// TwinCAT 3 PLC project Tc_Math
// Title: Tc_Math
// Company: NewEngineer
// Author: https://github.com/phucpha
// ProjectVersion: 0.0.0.1
// Description: this is library expand the Tc2_math
// ProgramVersion: 3.1.4024.0
// libraries:
//   Tc2_Standard, * (Beckhoff Automation GmbH)
//   Tc2_System, * (Beckhoff Automation GmbH)
//   Tc2_Utilities, * (Beckhoff Automation GmbH)
//   Tc3_Module, * (Beckhoff Automation GmbH)
// project tree:
//   DUTs/ E_CompareTime.TcDUT (not stored)
//   FCs/ F_CompareTime.TcPOU (not stored), FUN_Ceil.TcPOU (not stored), F_CheckInRange.TcPOU (not stored), F_CubicFit.TcPOU (not stored), F_CubitCalculate.TcPOU (not stored), F_InRange.TcPOU, F_QuanDraticCalculate.TcPOU (not stored), F_QuandraticFomularMaxValue.TcPOU (not stored), F_RoundLrealEx.TcPOU (not stored), F_ScaleValue.TcPOU (not stored)
//   / PlcTask.TcTTO (not stored)
//   POUs/ FB_CalCulateAccumulation.TcPOU (not stored), FB_Derivative.TcPOU

// ---- FCs/F_InRange.TcPOU
FUNCTION F_InRange : BOOL // return true if value in [bound1, bound2] or in [bound2, bound1] else return false
VAR_INPUT
	bound1 : LREAL;
	bound2 : LREAL;
	value	: LREAL;
END_VAR
VAR
END_VAR

F_InRange := (MIN(bound1, bound2) <= value)
				AND (value <= MAX(bound1, bound2));

END_FUNCTION

// ---- POUs/FB_Derivative.TcPOU
(*algorithm: Backward differentiation formula
the higher other the less stable , but more accuracy*)
FUNCTION_BLOCK FB_Derivative// unit : dentalvalue/seconde
VAR_INPUT
	bReset : BOOL	:= FALSE; //BOOL //reset
	lrInputValue : LREAL;// actual function value
	tDerivative	: TIME	:= T#1S; //length of time interval [tn−1,tn]  (equals time passed since last call to function)
	nOrder		: UINT := 3;// The s-step or order in algorithm // recommend
END_VAR
VAR_OUTPUT
	lrDerivative : LREAL;
	xValid : BOOL;//Validity OF result FALSE: If the number of calls neccessary for approximating has not been executed yet.
END_VAR
VAR
	ftn :LREAL;
	ftn_1 : LREAL;
	ftn_2 : LREAL;
	ftn_3 : LREAL;
	ftn_4 : LREAL;
	ftn_5	: LREAL;
	ftn_6	: LREAL;
	tonUpdate : TON;
	nTimeUpdate : LREAL;
END_VAR

IF bReset THEN
	tonUpdate.IN := FALSE;
	ftn := 0 ;
	ftn_1 := 0;
	ftn_2 := 0;
	ftn_3 := 0;
	ftn_4 := 0;
	ftn_5 := 0;
	ftn_6 := 0;
	nTimeUpdate := 0;
END_IF

tonUpdate( IN := TRUE,
			PT := tDerivative);
			
IF tonUpdate.Q THEN
	tonUpdate( IN := FALSE);
	ftn_6 := ftn_5;
	ftn_5 := ftn_4;
	ftn_4 := ftn_3;
	ftn_3 := ftn_2;
	ftn_2 := ftn_1;
	ftn_1 := ftn;
	ftn := lrInputValue;
	IF nTimeUpdate >= nOrder THEN
		nTimeUpdate := nOrder;
	ELSE 	
		nTimeUpdate := nTimeUpdate + 1;
	END_IF
END_IF
xValid := nTimeUpdate = nOrder;

IF tDerivative > T#0S THEN
	CASE nOrder OF
		1:  lrDerivative := (ftn - ftn_1)/ (TIME_TO_LREAL(tDerivative)/1000);
		2:  lrDerivative := (3*ftn - 4*ftn_1 + ftn_2)/ (2*TIME_TO_LREAL(tDerivative)/1000);
		3:	lrDerivative := (3*(ftn-ftn_3) + ftn_1 - ftn_2)/ (10*TIME_TO_LREAL(tDerivative)/1000);
		4:	lrDerivative :=	(25*ftn - 48*ftn_1 + 36*ftn_2 - 16*ftn_3 + 3*ftn_4)/ (12*TIME_TO_LREAL(tDerivative)/1000);
		5:	lrDerivative :=	(137*ftn - 300*ftn_1 + 300*ftn_2 - 200*ftn_3 + 75*ftn_4 - 12*ftn_5 )/(60*TIME_TO_LREAL(tDerivative)/1000);
		6:	lrDerivative :=	(147*ftn - 360*ftn_1 + 450*ftn_2 - 400*ftn_3 + 225*ftn_4 - 72*ftn_5 + 10*ftn_6)/(60*TIME_TO_LREAL(tDerivative)/1000);
	END_CASE
ELSE 
	lrDerivative := -8888888888888.4444;
	xValid := FALSE;
	
END_IF

END_FUNCTION_BLOCK
